// TIA Portal project "Paketleme Ve Paletleme" (V16)

(* hardware
DEVICE "S71500/ET200MP station_1"  S7-1500 station
   slot 0: "Rail_0"  Rack  6ES7 590-1***0-0AA0
   slot 1: "PLC_1"  CPU 1511-1 PN  6ES7 511-1AK02-0AB0  V2.8
      slot 3: "CPU display_1"  6ES7591-1AA00-0AA0
      slot 32768: "PROFINET interface_1"  X1
         slot 32769: "Port_1"  X1 P1
         slot 32770: "Port_2"  X1 P2
      slot 34817: "Virtual CP interface port_1"  Virtual CP interface port  Virtual CP interface port
   slot 2: "AI 8xU/I/RTD/TC ST_1"  AI 8xU/I/RTD/TC ST  6ES7 531-7KF00-0AB0  V2.0
   slot 3: "AI 8xU/I/RTD/TC ST_2"  AI 8xU/I/RTD/TC ST  6ES7 531-7KF00-0AB0  V2.0
   slot 4: "AI 8xU/I/RTD/TC ST_3"  AI 8xU/I/RTD/TC ST  6ES7 531-7KF00-0AB0  V2.0
   slot 5: "AI 8xU/I/RTD/TC ST_4"  AI 8xU/I/RTD/TC ST  6ES7 531-7KF00-0AB0  V2.0
   slot 6: "DI 16x24VDC BA_1"  DI 16x24VDC BA  6ES7 521-1BH10-0AA0  V1.0
   slot 7: "AI 8xU/I/RTD/TC ST_5"  AI 8xU/I/RTD/TC ST  6ES7 531-7KF00-0AB0  V2.0
   slot 8: "AI 8xU/I/RTD/TC ST_6"  AI 8xU/I/RTD/TC ST  6ES7 531-7KF00-0AB0  V2.0
   slot 9: "AI 8xU/I/RTD/TC ST_7"  AI 8xU/I/RTD/TC ST  6ES7 531-7KF00-0AB0  V2.0
   slot 10: "AQ 4xU/I ST_1"  AQ 4xU/I ST  6ES7 532-5HD00-0AB0  V2.0
   slot 11: "AQ 4xU/I ST_2"  AQ 4xU/I ST  6ES7 532-5HD00-0AB0  V2.0
   slot 12: "AQ 4xU/I ST_3"  AQ 4xU/I ST  6ES7 532-5HD00-0AB0  V2.0
   slot 13: "AQ 4xU/I ST_4"  AQ 4xU/I ST  6ES7 532-5HD00-0AB0  V2.0
   slot 14: "AQ 4xU/I ST_5"  AQ 4xU/I ST  6ES7 532-5HD00-0AB0  V2.0
   slot 15: "DQ 32x24VDC/0.5A BA_1"  DQ 32x24VDC/0.5A BA  6ES7 522-1BL10-0AA0  V1.0
   slot 16: "DI 32x24VDC BA_1"  DI 32x24VDC BA  6ES7 521-1BL10-0AA0  V1.0
*)

// ===== PLC "PLC_1"  CPU 1511-1 PN =====

VAR_GLOBAL   // PLC tag table "Default tag table"
   "Sistem Mem" AT %M90.0 : Bool;
END_VAR

VAR_GLOBAL   // PLC tag table "Inputs"
   "START BUTONU" AT %I0.0 : Bool;
   "STOP BUTONU" AT %I0.1 : Bool;
   "RESET BUTONU" AT %I0.2 : Bool;
   "MAVİ PİSTON İLERİDE" AT %I0.3 : Bool;
   "MAVİ PİSTON GERİDE" AT %I0.4 : Bool;
   "YEŞİL PİSTON İLERİDE" AT %I0.5 : Bool;
   "YEŞİL PİSTON GERİDE" AT %I0.6 : Bool;
   "GRİ PİSTON İLERİDE" AT %I0.7 : Bool;
   "GRİ PİSTON GERİDE" AT %I1.0 : Bool;
   "MAVİ ÜRÜN CNC GİRİŞ" AT %I1.1 : Bool;
   "YEŞİL ÜRÜN CNC GİRİŞ" AT %I1.2 : Bool;
   "GRİ ÜRÜN CNC GİRİŞ" AT %I1.3 : Bool;
   "MAVİ ÜRÜN CNC ÇIKIŞ" AT %I1.4 : Bool;
   "YEŞİL ÜRÜN CNC ÇIKIŞ" AT %I1.5 : Bool;
   "GRİ ÜRÜN CNC ÇIKIŞ" AT %I1.6 : Bool;
   "OGE İŞLENİYOR MAVİ" AT %I1.7 : Bool;
   "OGE İŞLENİYOR YEŞİL" AT %I2.0 : Bool;
   "OGE İŞLENİYOR GRİ" AT %I2.1 : Bool;
   "MAVİ ÜRÜN DÜZLEŞTİRİCİ SENSÖR" AT %I2.2 : Bool;
   "MAVİ KAPAK DÜZLEŞTİRİCİ SENSÖR" AT %I2.3 : Bool;
   "YEŞİL ÜRÜN DÜZLEŞTİRİCİ SENSÖR" AT %I2.4 : Bool;
   "YEŞİL  KAPAK DÜZLEŞTİRİCİ SENSÖR" AT %I2.5 : Bool;
   "GRİ ÜRÜN DÜZLEŞTİRİCİ SENSÖR" AT %I2.6 : Bool;
   "GRİ KAPAK DÜZLEŞTİRİCİ SENSÖR" AT %I2.7 : Bool;
   "MAVİ KAPAK DÜZLEŞTİRCİ AKTİF" AT %I3.0 : Bool;
   "MAVİ ÜRÜN DÜZLEŞTİRİCİ AKTİF" AT %I3.1 : Bool;
   "MAVİ DÜZLEŞTİRİCİ SON AKTİF" AT %I3.2 : Bool;
   "MAVİ ÜRÜN DÜZLEŞTİRİCİ LİMİT" AT %I3.3 : Bool;
   "YEŞİL  KAPAK DÜZLEŞTİRCİ AKTİF" AT %I3.4 : Bool;
   "YEŞİL  ÜRÜN DÜZLEŞTİRİCİ AKTİF" AT %I3.5 : Bool;
   "YEŞİL  DÜZLEŞTİRİCİ SON AKTİF" AT %I3.6 : Bool;
   "YEŞİL ÜRÜN DÜZLEŞTİRİCİ LİMİT" AT %I3.7 : Bool;
   "GRİ  KAPAK DÜZLEŞTİRCİ AKTİF" AT %I4.0 : Bool;
   "GRİ  ÜRÜN DÜZLEŞTİRİCİ AKTİF" AT %I4.1 : Bool;
   "GRİ  DÜZLEŞTİRİCİ SON AKTİF" AT %I4.2 : Bool;
   "GRİ ÜRÜN DÜZLEŞTİRİCİ LİMİT" AT %I4.3 : Bool;
   "MAVİ ROBOT-1 X AKTİF" AT %I4.4 : Bool;
   "MAVİ ROBOT-1 Z AKTİF" AT %I4.5 : Bool;
   "MAVİ ROBOT-1 TERSE DÖN AKTİF" AT %I4.6 : Bool;
   "MAVİ ROBOT-2 X AKTİF" AT %I4.7 : Bool;
   "MAVİ ROBOT-2 Z AKTİF" AT %I5.0 : Bool;
   "MAVİ ROBOT-2 TERSE DÖN AKTİF" AT %I5.1 : Bool;
   "YEŞİL ROBOT-1 X AKTİF" AT %I5.2 : Bool;
   "YEŞİL ROBOT-1 Z AKTİF" AT %I5.3 : Bool;
   "YEŞİL ROBOT-1 TERSE DÖN AKTİF" AT %I5.4 : Bool;
   "YEŞİL ROBOT-2 X AKTİF" AT %I5.5 : Bool;
   "YEŞİL ROBOT-2 Z AKTİF" AT %I5.6 : Bool;
   "YEŞİL ROBOT-2 TERSE DÖN AKTİF" AT %I5.7 : Bool;
   "GRİ ROBOT-1 X AKTİF" AT %I6.0 : Bool;
   "GRİ ROBOT-1 Z AKTİF" AT %I6.1 : Bool;
   "GRİ ROBOT-1 TERSE DÖN AKTİF" AT %I6.2 : Bool;
   "GRİ ROBOT-2 X AKTİF" AT %I6.3 : Bool;
   "GRİ ROBOT-2 Z AKTİF" AT %I6.4 : Bool;
   "GRİ ROBOT-2 TERSE DÖN AKTİF" AT %I6.5 : Bool;
   "KUTU-1 DURMA SENSÖRÜ NC" AT %I6.6 : Bool;
   "KUTU-2 DURMA SENSÖRÜ NC" AT %I6.7 : Bool;
   "KUTU-3 DURMA SENSÖRÜ NC" AT %I7.0 : Bool;
   "MAVİ SENSÖR" AT %I7.1 : Bool;
   "YEŞİL SENSÖR" AT %I7.2 : Bool;
   "GRİ SENSÖR" AT %I7.3 : Bool;
   "PL Piston-1 İleride" AT %I7.4 : Bool;
   "PL Piston-1 Geride" AT %I7.5 : Bool;
   "PL Piston-2 İleride" AT %I7.6 : Bool;
   "PL Piston-2 Geride" AT %I7.7 : Bool;
   "PL DONUS-1 İLERİ LİMİT" AT %I8.0 : Bool;
   "PL DONUS-1 GERİ LİMİT" AT %I8.1 : Bool;
   "PL DONUS-1 0 DA" AT %I8.2 : Bool;
   "PL DONUS-1 90 DA" AT %I8.3 : Bool;
   "PL DONUS-2 İLERİ LİMİT" AT %I8.4 : Bool;
   "PL DONUS-2 GERİ LİMİT" AT %I8.5 : Bool;
   "PL DONUS-2 0 DA" AT %I8.6 : Bool;
   "PL DONUS-2 90 DA" AT %I8.7 : Bool;
   "PL-1 PUSH LİMİT" AT %I9.0 : Bool;
   "PL-1 SIKIŞTIRMA AKTİF" AT %I9.1 : Bool;
   "PL-1 KAPAK KAPALI" AT %I9.2 : Bool;
   "PL-1 HARAKET EDİYOR" AT %I9.3 : Bool;
   "PL-2 PUSH LİMİT" AT %I9.4 : Bool;
   "PL-2 SIKIŞTIRMA AKTİF" AT %I9.5 : Bool;
   "PL-2 KAPAK KAPALI" AT %I9.6 : Bool;
   "PL-2 HARAKET EDİYOR" AT %I9.7 : Bool;
   "PL-1 DEPO ÜRÜN GİRİŞ" AT %I10.0 : Bool;
   "PL-2 DEPO ÜRÜN GİRİŞ" AT %I10.1 : Bool;
   "PL-1 PALET GİRİŞ" AT %I10.2 : Bool;
   "PL-2 PALET GİRİŞ" AT %I10.3 : Bool;
   "ANA PALET BESLEME SENSÖRÜ" AT %I10.4 : Bool;
END_VAR

VAR_GLOBAL   // PLC tag table "Outputs"
   "KONVEYOR-1" AT %Q0.0 : Bool;
   "KONVEYOR-2" AT %Q0.1 : Bool;
   "KONVEYOR-3" AT %Q0.2 : Bool;
   "MAVİ PİSTON" AT %Q0.3 : Bool;
   "YEŞİL PİSTON" AT %Q0.4 : Bool;
   "GRİ PİSTON" AT %Q0.5 : Bool;
   "MAVİ ÜRÜN KONVEYOR-1" AT %Q0.6 : Bool;
   "YEŞİL ÜRÜN KONVEYOR-1" AT %Q0.7 : Bool;
   "GRİ ÜRÜN KONVEYOR-1" AT %Q1.0 : Bool;
   "MAVİ CNC" AT %Q1.1 : Bool;
   "YEŞİL CNC" AT %Q1.2 : Bool;
   "GRİ CNC" AT %Q1.3 : Bool;
   "MAVİ ÜRÜN KONVEYOR-2" AT %Q1.4 : Bool;
   "MAVİ KAPAK KONVEYOR" AT %Q1.5 : Bool;
   "KUTU KONVEYOR-1" AT %Q1.6 : Bool;
   "YEŞİL ÜRÜN KONVEYOR-2" AT %Q1.7 : Bool;
   "YEŞİL KAPAK KONVEYOR" AT %Q2.0 : Bool;
   "KUTU KONVEYOR-2" AT %Q2.1 : Bool;
   "GRİ ÜRÜN KONVEYOR-2" AT %Q2.2 : Bool;
   "GRİ KAPAK KONVEYOR" AT %Q2.3 : Bool;
   "KUTU KONVEYOR-3" AT %Q2.4 : Bool;
   "MAVİ ÜRÜN DÜZLEŞTİRİCİ" AT %Q2.5 : Bool;
   "MAVİ KAPAK DÜZLEŞTİRİCİ" AT %Q2.6 : Bool;
   "MAVİ DÜZLEŞTRİCİ SON" AT %Q2.7 : Bool;
   "YEŞİL ÜRÜN DÜZLEŞTİRİCİ" AT %Q3.0 : Bool;
   "YEŞİL KAPAK DÜZLEŞTİRİCİ" AT %Q3.1 : Bool;
   "YEŞİL DÜZLEŞTRİCİ SON" AT %Q3.2 : Bool;
   "GRİ ÜRÜN DÜZLEŞTİRİCİ" AT %Q3.3 : Bool;
   "GRİ KAPAK DÜZLEŞTİRİCİ" AT %Q3.4 : Bool;
   "GRİ DÜZLEŞTRİCİ SON" AT %Q3.5 : Bool;
   "MAVİ ROBOT-1 X GİT" AT %Q3.6 : Bool;
   "MAVİ ROBOT-1 Z GİT" AT %Q3.7 : Bool;
   "MAVİ ROBOT-1 VAKUM AÇ" AT %Q4.0 : Bool;
   "MAVİ ROBOT-1 TERSE DÖN" AT %Q4.1 : Bool;
   "MAVİ ROBOT-2 X GİT" AT %Q4.2 : Bool;
   "MAVİ ROBOT-2 Z GİT" AT %Q4.3 : Bool;
   "MAVİ ROBOT-2 VAKUM AÇ" AT %Q4.4 : Bool;
   "MAVİ ROBOT-2 TERSE DÖN" AT %Q4.5 : Bool;
   "YEŞİL  ROBOT-1 X GİT" AT %Q4.6 : Bool;
   "YEŞİL ROBOT-1 Z GİT" AT %Q4.7 : Bool;
   "YEŞİL ROBOT-1 VAKUM AÇ" AT %Q5.0 : Bool;
   "YEŞİL ROBOT-1 TERSE DÖN" AT %Q5.1 : Bool;
   "YEŞİL ROBOT-2 X GİT" AT %Q5.2 : Bool;
   "YEŞİL ROBOT-2 Z GİT" AT %Q5.3 : Bool;
   "YEŞİL ROBOT-2 VAKUM AÇ" AT %Q5.4 : Bool;
   "YEŞİL ROBOT-2 TERSE DÖN" AT %Q5.5 : Bool;
   "GRİ  ROBOT-1 X GİT" AT %Q5.6 : Bool;
   "GRİ ROBOT-1 Z GİT" AT %Q5.7 : Bool;
   "GRİ ROBOT-1 VAKUM AÇ" AT %Q6.0 : Bool;
   "GRİ ROBOT-1 TERSE DÖN" AT %Q6.1 : Bool;
   "GRİ ROBOT-2 X GİT" AT %Q6.2 : Bool;
   "GRİ ROBOT-2 Z GİT" AT %Q6.3 : Bool;
   "GRİ ROBOT-2 VAKUM AÇ" AT %Q6.4 : Bool;
   "YEŞİL ROBOT-2 TERSE DÖN(1)" AT %Q6.5 : Bool;
   "MAVİ DÜZLEŞTİRCİ YUKARI" AT %Q6.6 : Bool;
   "YEŞİL DÜZLEŞTİRCİ YUKARI" AT %Q6.7 : Bool;
   "GRİ DÜZLEŞTİRCİ YUKARI" AT %Q7.0 : Bool;
   "GRİ DEPO KONVEYORU-1" AT %Q7.1 : Bool;
   "GRİ DEPO KONVEYORU-2" AT %Q7.2 : Bool;
   "GRİ DEPO KONVEYORU-3" AT %Q7.3 : Bool;
   "YEŞİL DEPO KONVEYORU-1" AT %Q7.4 : Bool;
   "YEŞİL DEPO KONVEYORU-2" AT %Q7.5 : Bool;
   "DONUS-1 İLERİ" AT %Q7.6 : Bool;
   "DONUS-1 GERİ" AT %Q7.7 : Bool;
   "DONUS-1 DONDUR" AT %Q8.0 : Bool;
   "DONUS-2 İLERİ" AT %Q8.1 : Bool;
   "DONUS-2 GERİ" AT %Q8.2 : Bool;
   "DONUS-2 DONDRU" AT %Q8.3 : Bool;
   "DEPO KONVEYOR-1" AT %Q8.4 : Bool;
   "DEPO KONVEYOR-2" AT %Q8.5 : Bool;
   "DEPO KONVEYOR-3" AT %Q8.6 : Bool;
   "PL Piston-1" AT %Q8.7 : Bool;
   "PL Piston-2" AT %Q9.0 : Bool;
   "PL KONVEYOR-1" AT %Q9.1 : Bool;
   "PL KONVEYOR-2" AT %Q9.2 : Bool;
   "PL KONVEYOR-3" AT %Q9.3 : Bool;
   "PL KONVEYOR-4" AT %Q9.4 : Bool;
   "PL KONVEYOR-5" AT %Q9.5 : Bool;
   "PL KONVEYOR-6" AT %Q9.6 : Bool;
   "PL KONVEYOR-7" AT %Q9.7 : Bool;
   "PL KONVEYOR-8" AT %Q10.0 : Bool;
   "PALET BESLEME KONVEYOR-1" AT %Q10.1 : Bool;
   "PALET KONVEYOR-2" AT %Q10.2 : Bool;
   "PALET KONVEYOR-3" AT %Q10.3 : Bool;
   "PALET KONVEYOR-4" AT %Q10.4 : Bool;
   "PALET KONVEYOR-5" AT %Q10.5 : Bool;
   "PALET KONVEYOR-6" AT %Q10.6 : Bool;
   "PALET KONVEYOR-7" AT %Q10.7 : Bool;
   "PALET KONVEYOR-8" AT %Q11.0 : Bool;
   "PALET KONVEYOR-9" AT %Q11.1 : Bool;
   "PL DONUS-1 İLERİ" AT %Q11.2 : Bool;
   "PL DONUS-1 GERİ" AT %Q11.3 : Bool;
   "PL DONUS-1" AT %Q11.4 : Bool;
   "PL DONUS-2 İLERİ" AT %Q11.5 : Bool;
   "PL DONUS-2 GERİ" AT %Q11.6 : Bool;
   "PL DONUS-2" AT %Q11.7 : Bool;
   "Palet Depo Konveypru-1" AT %Q12.0 : Bool;
   "Palet Depo Konveypru-2" AT %Q12.1 : Bool;
   "Palet Depo Konveypru-3" AT %Q12.2 : Bool;
   "Palet Depo Konveypru-4" AT %Q12.3 : Bool;
   "Palet Depo Konveypru-5" AT %Q12.4 : Bool;
   "Palet Depo Konveypru-6" AT %Q12.5 : Bool;
   "Palet Depo Konveypru-7" AT %Q12.6 : Bool;
   "Palet Depo Konveypru-8" AT %Q12.7 : Bool;
   "PL-1 ÜST GERİ" AT %Q13.0 : Bool;
   "PL-1 ÜST İLERİ" AT %Q13.1 : Bool;
   "PL-1 DÜZLEŞTİRME" AT %Q13.2 : Bool;
   "PL-1 PUSH" AT %Q13.3 : Bool;
   "PL-1 KAPAK AÇMA" AT %Q13.4 : Bool;
   "PL-1 SIKIŞTIRMA" AT %Q13.5 : Bool;
   "PL-1 ALT İLERİ" AT %Q13.6 : Bool;
   "PL-1 ALT GERİ" AT %Q13.7 : Bool;
   "PL-1 AŞŞAĞI" AT %Q14.0 : Bool;
   "PL-1 YUKARI" AT %Q14.1 : Bool;
   "PL-1 YUKARI LİMİTE ÇIK" AT %Q14.2 : Bool;
   "PL-2 ÜST GERİ" AT %Q14.3 : Bool;
   "PL-2 ÜST İLERİ" AT %Q14.4 : Bool;
   "PL-2 DÜZLEŞTİRME" AT %Q14.5 : Bool;
   "PL-2 PUSH" AT %Q14.6 : Bool;
   "PL-2 KAPAK AÇMA" AT %Q14.7 : Bool;
   "PL-2 SIKIŞTIRMA" AT %Q15.0 : Bool;
   "PL-2 ALT İLERİ" AT %Q15.1 : Bool;
   "PL-2 ALT GERİ" AT %Q15.2 : Bool;
   "PL-2 AŞŞAĞI" AT %Q15.3 : Bool;
   "PL-2 YUKARI" AT %Q15.4 : Bool;
   "PL-2 YUKARI LİMİTE ÇIK" AT %Q15.5 : Bool;
END_VAR

FUNCTION "Sistem Start" : Void   // FC1, LAD
{ S7_Optimized_Access := 'TRUE' }
VERSION : 0.1
BEGIN

REGION Network 1: SİSTEM START
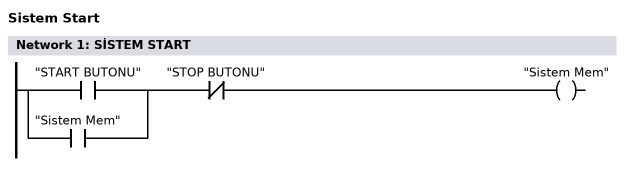
   RUNG wire#powerrail
      Contact( "START BUTONU" )
      wire#w1
      I_Contact( "STOP BUTONU" )
      Coil( "Sistem Mem" )
   END_RUNG
   RUNG wire#powerrail
      Contact( "Sistem Mem" )
   END_RUNG wire#w1
   // the same network as SCL:
   "Sistem Mem" := ("START BUTONU" OR "Sistem Mem") AND NOT "STOP BUTONU";
END_REGION
END_FUNCTION

FUNCTION "MHJ-PLC-Lab-Function-S71500" : Void   // FC9000, SCL
{ S7_Optimized_Access := 'TRUE' }
VERSION : 0.1
   VAR_TEMP
      Value : Byte;
      ForCounter : Int;
   END_VAR
   VAR CONSTANT
      Value_01_DW : DWord := 16#1223_5486;
      Value_02_DW : DWord := 16#A6C9_D1F5;
   END_VAR
BEGIN

   #Value:=PEEK(area := 16#82,
        dbNumber := 0,
        byteOffset := 511);
   #Value := #Value + 1;

   POKE(area := 16#82,
        dbNumber := 0,
        byteOffset := 511,
        value := #Value);

   POKE(area := 16#82,
        dbNumber := 0,
        byteOffset := 1016,
        value := #Value_01_DW);
   POKE(area := 16#82,
        dbNumber := 0,
        byteOffset := 1020,
        value := #Value_02_DW);

   FOR #ForCounter := 0 TO 63 DO
       #Value:=PEEK(area := 16#1,
            dbNumber := 0,
            byteOffset := #ForCounter);
       POKE(area := 16#81,
            dbNumber := 0,
            byteOffset := #ForCounter,
            value := #Value);
   END_FOR;
   #Value := PEEK(area := 16#1,
                  dbNumber := 0,
                  byteOffset := 512);
   POKE(area := 16#82,
        dbNumber := 0,
        byteOffset := 512,
        value := #Value);
END_FUNCTION

ORGANIZATION_BLOCK "Main"   // OB1, LAD, ProgramCycle
TITLE = "Main Program Sweep (Cycle)"
{ S7_Optimized_Access := 'TRUE' }
VERSION : 0.1
   VAR_INPUT
      Initial_Call : Bool;   // Initial call of this OB
      Remanence : Bool;   // =True, if remanent data are available
   END_VAR
BEGIN

REGION Network 1: PLC - FACTORYIO CONN
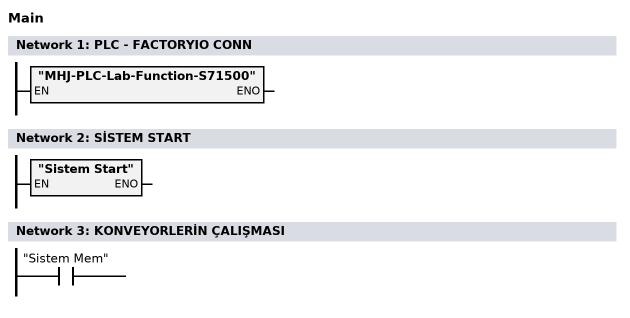
   RUNG wire#powerrail
      "MHJ-PLC-Lab-Function-S71500"()
   END_RUNG
   // the same network as SCL:
   "MHJ-PLC-Lab-Function-S71500"();
END_REGION

REGION Network 2: SİSTEM START
   RUNG wire#powerrail
      "Sistem Start"()
   END_RUNG
   // the same network as SCL:
   "Sistem Start"();
END_REGION

REGION Network 3: KONVEYORLERİN ÇALIŞMASI
END_REGION
END_ORGANIZATION_BLOCK